
// ===== library: MasterCopy "BVS_Sensor" =====

FUNCTION_BLOCK "BVS_Sensor"   // FB52, SCL
TITLE = BVS_ID
{ S7_Optimized_Access := 'FALSE' }
AUTHOR : PD-ILS
FAMILY : Balluff
VERSION : 1.1
// Functionblock for BVS ID and BVS VS.
// Compatible with Profinet and IO-Link version.
BEGIN
END_FUNCTION_BLOCK